// TIA Portal V16 export
// export: Created 2021-11-12T13:31:51.744499Z, ExportSetting WithDefaults, DisplayName Totally Integrated Automation Portal, DisplayVersion V16 Update 3, DisplayName TIA Portal Version Control Interface, DisplayVersion V16 Update 2, DisplayName TIA Portal Openness, DisplayVersion V16 Update 3, DisplayName SINAMICS Startdrive Advanced, DisplayVersion V16 Update 5, DisplayName SINAMICS Startdrive G130, G150, S120, S150, SINAMICS MV, S210, DisplayVersion V16 Update 5, DisplayName SINAMICS Startdrive G110M, G120, G120C, G120D, G120P, G115D, DisplayVersion V16 Update 5, DisplayName STEP 7 Professional, DisplayVersion V16 Update 3, DisplayName STEP 7 Safety, DisplayVersion V16, DisplayName WinCC UA Professional, DisplayVersion V16 Update 3
DATA_BLOCK "STATUS_000+UH01"   // DB2022
{ S7_Optimized_Access := 'TRUE' }
VERSION : 0.1
// stored: AutoNumber false, DBAccessibleFromOPCUA true, IsOnlyStoredInLoadMemory false, IsRetainMemResEnabled false, IsWriteProtectedInAS false, MemoryReserve 100
   VAR
      xxxxx___BinarySensors___xxxxx : Byte;
      xxxxx___BinaryOthers___xxxxx : Byte;
      "UC01-FV01_11" : Bool;   // Přepěťová ochrana OK
      "UC01-FC01_14" : Bool;   // Osvětlení a zásuvky 230V Nadproudová ochrana OK
      "UC01-FB01_14" : Bool;   // Osvětlení a zásuvky 230V Napájecí a řídící rozvaděč OK
      "I100.3" : Bool;   // Rezerva
      "I100.4" : Bool;   // Rezerva
      "I100.5" : Bool;   // Rezerva
      "I100.6" : Bool;   // Rezerva
      "I100.7" : Bool;   // Rezerva
      "100UC01-FC21_14" : Bool;   // Napájení klimatizace Hlavní rozvaděč OK
      "UC01-EC01_14" : Bool;   // Chlazení rozvaděče OK
      "UC01-FC22_14" : Bool;   // Napájení 230V Centrální pult OK
      "UC01-FC23_14" : Bool;   // Napájení klimatizace Centrální pult OK
      "UC01-FC24_14" : Bool;   // Napájení klimatizace Centrální panel OK
      "400UC01-FC21_14" : Bool;   // Napájení Osvětlení kamer OK
      "400UC01-FC22_14" : Bool;   // Napájení Ventily Memtech OK
      "I101.7" : Bool;   // Rezerva
      "UH01-FC30_14" : Bool;   // 24VDC (UPS) Jištění OK
      "UH01-FC30_24" : Bool;   // 24VDC (UPS) Zatížení < 90% OK
      "UC01-RB01_24" : Bool;   // UPS Baterie OK
      "UH01-FC50_14" : Bool;   // 24VDC Jištění OK
      "UH01-FC50_24" : Bool;   // 24VDC Zatížení < 90% OK
      "I102.5" : Bool;   // Rezerva
      "I102.6" : Bool;   // Rezerva
      "I102.7" : Bool;   // Rezerva
      xxxxx___InterfaceSignals___xxxxx : Byte;
      SumErr : Bool;   // Sum of significant errors
      PwrOK : Bool;   // Significant switches ON
      xxxxx___AnalogueSensors___xxxxx : Byte;
      xxxxx___Drives___xxxxx : Byte;
      xxxxx___Other___xxxxx : Byte;
      xxxxx__Alarms___xxxxx : Byte;
      "UC01-FV01_12" : Struct   // Surge suppressor is OK / Přepěťová ochrana OK
         Main { S7_SetPoint := 'True'} : "UDT_Status_main";
         Specific { S7_SetPoint := 'True'} : "UDT_DI_Mon_Status_specific";
         Error { S7_SetPoint := 'True'} : "UDT_Error01";
      END_STRUCT;
      "UC01-FC01_15" : Struct   // Light & socket 230V overcurrent protection is OK / Osvětlení a zásuvky 230V Nadproudová ochrana OK
         Main { S7_SetPoint := 'True'} : "UDT_Status_main";
         Specific { S7_SetPoint := 'True'} : "UDT_DI_Mon_Status_specific";
         Error { S7_SetPoint := 'True'} : "UDT_Error01";
      END_STRUCT;
      "UC01-FB01_15" : Struct   // Light & socket 230V main distributor is OK / Osvětlení a zásuvky 230V Napájecí a řídící rozvaděč OK
         Main { S7_SetPoint := 'True'} : "UDT_Status_main";
         Specific { S7_SetPoint := 'True'} : "UDT_DI_Mon_Status_specific";
         Error { S7_SetPoint := 'True'} : "UDT_Error01";
      END_STRUCT;
      "I100.8" : Struct   // Rezerva
         Main { S7_SetPoint := 'True'} : "UDT_Status_main";
         Specific { S7_SetPoint := 'True'} : "UDT_DI_Mon_Status_specific";
         Error { S7_SetPoint := 'True'} : "UDT_Error01";
      END_STRUCT;
      "I100.9" : Struct   // Rezerva
         Main { S7_SetPoint := 'True'} : "UDT_Status_main";
         Specific { S7_SetPoint := 'True'} : "UDT_DI_Mon_Status_specific";
         Error { S7_SetPoint := 'True'} : "UDT_Error01";
      END_STRUCT;
      "I100.10" : Struct   // Rezerva
         Main { S7_SetPoint := 'True'} : "UDT_Status_main";
         Specific { S7_SetPoint := 'True'} : "UDT_DI_Mon_Status_specific";
         Error { S7_SetPoint := 'True'} : "UDT_Error01";
      END_STRUCT;
      "I100.11" : Struct   // Rezerva
         Main { S7_SetPoint := 'True'} : "UDT_Status_main";
         Specific { S7_SetPoint := 'True'} : "UDT_DI_Mon_Status_specific";
         Error { S7_SetPoint := 'True'} : "UDT_Error01";
      END_STRUCT;
      "I100.12" : Struct   // Rezerva
         Main { S7_SetPoint := 'True'} : "UDT_Status_main";
         Specific { S7_SetPoint := 'True'} : "UDT_DI_Mon_Status_specific";
         Error { S7_SetPoint := 'True'} : "UDT_Error01";
      END_STRUCT;
      "100UC01-FC21_15" : Struct   // Power supply cooling Main distributor is OK / Napájení klimatizace Hlavní rozvaděč OK
         Main { S7_SetPoint := 'True'} : "UDT_Status_main";
         Specific { S7_SetPoint := 'True'} : "UDT_DI_Mon_Status_specific";
         Error { S7_SetPoint := 'True'} : "UDT_Error01";
      END_STRUCT;
      "UC01-EC01_15" : Struct   // Distributor cooling is OK / Chlazení rozvaděče OK
         Main { S7_SetPoint := 'True'} : "UDT_Status_main";
         Specific { S7_SetPoint := 'True'} : "UDT_DI_Mon_Status_specific";
         Error { S7_SetPoint := 'True'} : "UDT_Error01";
      END_STRUCT;
      "UC01-FC22_15" : Struct   // Power supply 230V Central pult OK / Napájení 230V Centrální pult OK
         Main { S7_SetPoint := 'True'} : "UDT_Status_main";
         Specific { S7_SetPoint := 'True'} : "UDT_DI_Mon_Status_specific";
         Error { S7_SetPoint := 'True'} : "UDT_Error01";
      END_STRUCT;
      "UC01-FC23_15" : Struct   // Power supply cooling Central panel is OK / Napájení klimatizace Centrální pult OK
         Main { S7_SetPoint := 'True'} : "UDT_Status_main";
         Specific { S7_SetPoint := 'True'} : "UDT_DI_Mon_Status_specific";
         Error { S7_SetPoint := 'True'} : "UDT_Error01";
      END_STRUCT;
      "UC01-FC24_15" : Struct   // Power supply cooling Central panel is OK / Napájení klimatizace Centrální panel OK
         Main { S7_SetPoint := 'True'} : "UDT_Status_main";
         Specific { S7_SetPoint := 'True'} : "UDT_DI_Mon_Status_specific";
         Error { S7_SetPoint := 'True'} : "UDT_Error01";
      END_STRUCT;
      "400UC01-FC21_15" : Struct   // Power supply cooling Camera light is OK / Napájení Osvětlení kamer OK
         Main { S7_SetPoint := 'True'} : "UDT_Status_main";
         Specific { S7_SetPoint := 'True'} : "UDT_DI_Mon_Status_specific";
         Error { S7_SetPoint := 'True'} : "UDT_Error01";
      END_STRUCT;
      "400UC01-FC22_15" : Struct   // Rezerva
         Main { S7_SetPoint := 'True'} : "UDT_Status_main";
         Specific { S7_SetPoint := 'True'} : "UDT_DI_Mon_Status_specific";
         Error { S7_SetPoint := 'True'} : "UDT_Error01";
      END_STRUCT;
      "I101.8" : Struct   // Rezerva
         Main { S7_SetPoint := 'True'} : "UDT_Status_main";
         Specific { S7_SetPoint := 'True'} : "UDT_DI_Mon_Status_specific";
         Error { S7_SetPoint := 'True'} : "UDT_Error01";
      END_STRUCT;
      "UH01-FC30_15" : Struct   // 24VDC (UPS) Protection is OK / 24VDC (UPS) Jištění OK
         Main { S7_SetPoint := 'True'} : "UDT_Status_main";
         Specific { S7_SetPoint := 'True'} : "UDT_DI_Mon_Status_specific";
         Error { S7_SetPoint := 'True'} : "UDT_Error01";
      END_STRUCT;
      "UH01-FC30_25" : Struct   // 24VDC (UPS) Load < 90% OK / 24VDC (UPS) Zatížení < 90% OK
         Main { S7_SetPoint := 'True'} : "UDT_Status_main";
         Specific { S7_SetPoint := 'True'} : "UDT_DI_Mon_Status_specific";
         Error { S7_SetPoint := 'True'} : "UDT_Error01";
      END_STRUCT;
      "UC01-RB01_25" : Struct   // UPS Battery is OK / UPS Baterie OK
         Main { S7_SetPoint := 'True'} : "UDT_Status_main";
         Specific { S7_SetPoint := 'True'} : "UDT_DI_Mon_Status_specific";
         Error { S7_SetPoint := 'True'} : "UDT_Error01";
      END_STRUCT;
      "UH01-FC50_15" : Struct   // 24VDC Protection is OK / 24VDC Jištění OK
         Main { S7_SetPoint := 'True'} : "UDT_Status_main";
         Specific { S7_SetPoint := 'True'} : "UDT_DI_Mon_Status_specific";
         Error { S7_SetPoint := 'True'} : "UDT_Error01";
      END_STRUCT;
      "UH01-FC50_25" : Struct   // 24VDC Load < 90% is OK / 24VDC Zatížení < 90% OK
         Main { S7_SetPoint := 'True'} : "UDT_Status_main";
         Specific { S7_SetPoint := 'True'} : "UDT_DI_Mon_Status_specific";
         Error { S7_SetPoint := 'True'} : "UDT_Error01";
      END_STRUCT;
      "I102.8" : Struct   // Rezerva
         Main { S7_SetPoint := 'True'} : "UDT_Status_main";
         Specific { S7_SetPoint := 'True'} : "UDT_DI_Mon_Status_specific";
         Error { S7_SetPoint := 'True'} : "UDT_Error01";
      END_STRUCT;
      "I102.9" : Struct   // Rezerva
         Main { S7_SetPoint := 'True'} : "UDT_Status_main";
         Specific { S7_SetPoint := 'True'} : "UDT_DI_Mon_Status_specific";
         Error { S7_SetPoint := 'True'} : "UDT_Error01";
      END_STRUCT;
      "I102.10" : Struct   // Rezerva
         Main { S7_SetPoint := 'True'} : "UDT_Status_main";
         Specific { S7_SetPoint := 'True'} : "UDT_DI_Mon_Status_specific";
         Error { S7_SetPoint := 'True'} : "UDT_Error01";
      END_STRUCT;
      ES : Struct   // E-stop
         Main { S7_SetPoint := 'True'} : "UDT_Status_main";
         Specific { S7_SetPoint := 'True'} : "UDT_DI_Mon_Status_specific";
         Error { S7_SetPoint := 'True'} : "UDT_Error01";
      END_STRUCT;
      "000UH01-KF31" : Struct   // Module 00UH01- KF31 / Modul 00UH01- KF31
         Main { S7_SetPoint := 'True'} : "UDT_Status_main";
         Specific { S7_SetPoint := 'True'} : "UDT_DI_Mon_Status_specific";
         Error { S7_SetPoint := 'True'} : "UDT_Error01";
      END_STRUCT;
      "000UH01-KF32" : Struct   // Module 00UH01- KF32 / Modul 00UH01- KF32
         Main { S7_SetPoint := 'True'} : "UDT_Status_main";
         Specific { S7_SetPoint := 'True'} : "UDT_DI_Mon_Status_specific";
         Error { S7_SetPoint := 'True'} : "UDT_Error01";
      END_STRUCT;
      "000UH01-KF33" : Struct   // Module 00UH01- KF33 / Modul 00UH01- KF33
         Main { S7_SetPoint := 'True'} : "UDT_Status_main";
         Specific { S7_SetPoint := 'True'} : "UDT_DI_Mon_Status_specific";
         Error { S7_SetPoint := 'True'} : "UDT_Error01";
      END_STRUCT;
      "000UH01-KF41" : Struct   // Module 00UH01- KF41 / Modul 00UH01- KF41
         Main { S7_SetPoint := 'True'} : "UDT_Status_main";
         Specific { S7_SetPoint := 'True'} : "UDT_DI_Mon_Status_specific";
         Error { S7_SetPoint := 'True'} : "UDT_Error01";
      END_STRUCT;
   END_VAR
BEGIN
END_DATA_BLOCK
